% RSLogix 500 project LIFT_0_BAK000.RSS, saved by version 7.30.10.01 %
PROJECT "LIFT_0"    % processor: type code 158 %

PROGRAM FILES
  LAD 2   7 rungs

DATA FILES
  O0 OUTPUT  186 elements
  I1 INPUT  130 elements
  S2 STATUS  83 elements
  B3 BINARY  1 elements
  T4 TIMER  1 elements
  C5 COUNTER  1 elements
  R6 CONTROL  1 elements
  N7 INTEGER  1 elements
  F8 FLOAT  1 elements

LADDER 2
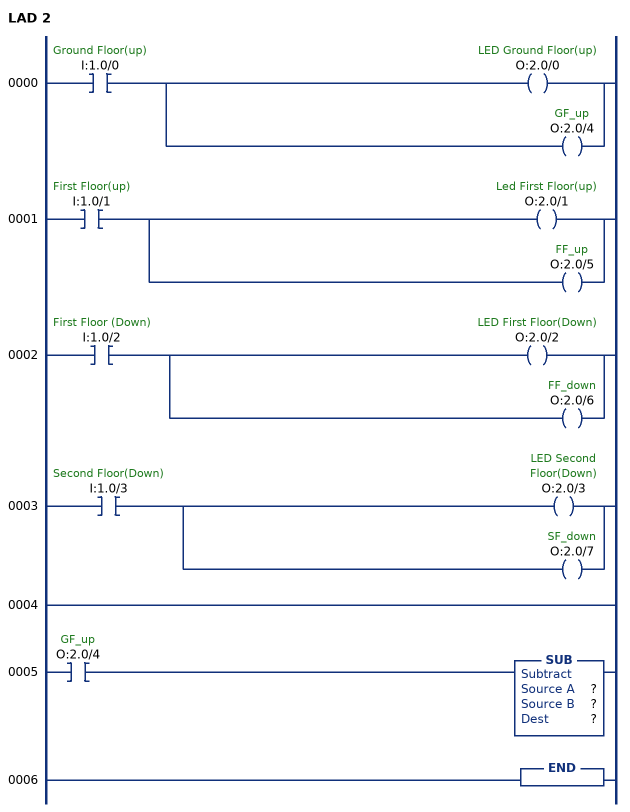
% Rung: 0 %  % edit flag set %
SOR XIC I:1.0/0 BST OTE O:2.0/0 NXB OTE O:2.0/4 BND EOR
%   I:1.0/0  "Ground Floor(up)" %
%   O:2.0/0  "LED Ground Floor(up)" %
%   O:2.0/4  "GF_up" %
% Rung: 1 %  % edit flag set %
SOR XIC I:1.0/1 BST OTE O:2.0/1 NXB OTE O:2.0/5 BND EOR
%   I:1.0/1  "First Floor(up)" %
%   O:2.0/1  "Led First Floor(up)" %
%   O:2.0/5  "FF_up" %
% Rung: 2 %  % edit flag set %
SOR XIC I:1.0/2 BST OTE O:2.0/2 NXB OTE O:2.0/6 BND EOR
%   I:1.0/2  "First Floor (Down)" %
%   O:2.0/2  "LED First Floor(Down)" %
%   O:2.0/6  "FF_down" %
% Rung: 3 %  % edit flag set %
SOR XIC I:1.0/3 BST OTE O:2.0/3 NXB OTE O:2.0/7 BND EOR
%   I:1.0/3  "Second Floor(Down)" %
%   O:2.0/3  "LED Second Floor(Down)" %
%   O:2.0/7  "SF_down" %
% Rung: 4 %  % edit flag set %
SOR EOR
% Rung: 5 %  % edit flag set %
SOR XIC O:2.0/4 SUB ? ? ? EOR
%   O:2.0/4  "GF_up" %
% Rung: 6 %
SOR END EOR

OTHER DOCUMENTED ADDRESSES
  N7:0  "Lift Current Floor"
